INTERFACE I_MotionLogger

METHOD Clear
VAR_INPUT
END_VAR
END_METHOD

METHOD ErrorCodeLookup : STRING
VAR_INPUT
	 nErrorId: UDINT;
END_VAR
END_METHOD

METHOD GetAllMessages : STRING(1024)
END_METHOD

METHOD GetMessageCount : UINT
VAR_OUTPUT
    nCount : UINT;
END_VAR
END_METHOD

METHOD Logger
VAR_INPUT
    Message : STRING;
    Level   : E_MotionLogLevel := E_MotionLogLevel.INFO;
    Source  : STRING := '';
END_VAR
END_METHOD

PROPERTY Name : STRING
GET
END_GET
END_PROPERTY

END_INTERFACE

(* stored: Version 1.1.0.1
   Itf I_MotionLogger: Id {ba839cec-9291-4692-8f1c-76e0f27d3db4}
   Method Clear: Id {7bbc559f-d817-41f1-8220-7fbb6113d4af}
   Method ErrorCodeLookup: Id {55ed6a2c-beff-40b2-b277-6cb853ad11a8}
   Method GetAllMessages: Id {0d8456d8-a972-467e-aec8-f7544ecc3e0f}
   Method GetMessageCount: Id {96dae5b2-bee3-4a4a-af42-11e4dbc3e083}
   Method Logger: Id {d06a0d50-48f4-4261-869e-95d5c3b0e14a}
   Property Name: Id {6e33c188-92bc-4132-b7e8-d2172b8babf5}
   Get Get: Id {9b2948a7-ea61-4c72-84b2-8ff692b52f06} *)
